      HW_2374P1_Interface_Port_1 { ExternalAccessible := 'False'; ExternalVisible := 'False'; ExternalWritable := 'False'} : HW_INTERFACE := 995;   // "2374P1~Interface~Port_1"
      HW_2374P1_Interface_Port_2 { ExternalAccessible := 'False'; ExternalVisible := 'False'; ExternalWritable := 'False'} : HW_INTERFACE := 996;   // "2374P1~Interface~Port_2"
      HW_2374P1_Head { ExternalAccessible := 'False'; ExternalVisible := 'False'; ExternalWritable := 'False'} : HW_SUBMODULE := 997;   // "2374P1~Head"
      HW_2374P1_EO_Multiturn_1 { ExternalAccessible := 'False'; ExternalVisible := 'False'; ExternalWritable := 'False'} : HW_SUBMODULE := 998;   // "2374P1~EO_Multiturn_1"
      HW_2374P1_Telegram_81_DI_DO { ExternalAccessible := 'False'; ExternalVisible := 'False'; ExternalWritable := 'False'} : HW_SUBMODULE := 999;   // "2374P1_Telegram_81~DI_DO"
      HW_2374P1_EO_Multiturn_1_Parameter_Access_Point { ExternalAccessible := 'False'; ExternalVisible := 'False'; ExternalWritable := 'False'} : HW_SUBMODULE := 1000;   // "2374P1~EO_Multiturn_1~Parameter_Access_Point"
      HW_100A1_Proxy { ExternalAccessible := 'False'; ExternalVisible := 'False'; ExternalWritable := 'False'} : HW_SUBMODULE := 866;   // "100A1~Proxy"
      HW_100A1_IODevice { ExternalAccessible := 'False'; ExternalVisible := 'False'; ExternalWritable := 'False'} : HW_DEVICE := 864;   // "100A1~IODevice"
      HW_100A1_PN_IO { ExternalAccessible := 'False'; ExternalVisible := 'False'; ExternalWritable := 'False'} : HW_INTERFACE := 867;   // "100A1~PN-IO"
      HW_100A1_PN_IO_Port_1 { ExternalAccessible := 'False'; ExternalVisible := 'False'; ExternalWritable := 'False'} : HW_INTERFACE := 868;   // "100A1~PN-IO~Port_1"
      HW_100A1_PN_IO_Port_2 { ExternalAccessible := 'False'; ExternalVisible := 'False'; ExternalWritable := 'False'} : HW_INTERFACE := 869;   // "100A1~PN-IO~Port_2"
      HW_100A1_Head { ExternalAccessible := 'False'; ExternalVisible := 'False'; ExternalWritable := 'False'} : HW_SUBMODULE := 870;   // "100A1~Head"
      HW_2394P1_Proxy { ExternalAccessible := 'False'; ExternalVisible := 'False'; ExternalWritable := 'False'} : HW_SUBMODULE := 1003;   // "2394P1~Proxy"
      HW_2394P1_IODevice { ExternalAccessible := 'False'; ExternalVisible := 'False'; ExternalWritable := 'False'} : HW_DEVICE := 1001;   // "2394P1~IODevice"
      HW_2394P1_Interface { ExternalAccessible := 'False'; ExternalVisible := 'False'; ExternalWritable := 'False'} : HW_INTERFACE := 1004;   // "2394P1~Interface"
      HW_2394P1_Interface_Port_1 { ExternalAccessible := 'False'; ExternalVisible := 'False'; ExternalWritable := 'False'} : HW_INTERFACE := 1005;   // "2394P1~Interface~Port_1"
      HW_2394P1_Interface_Port_2 { ExternalAccessible := 'False'; ExternalVisible := 'False'; ExternalWritable := 'False'} : HW_INTERFACE := 1006;   // "2394P1~Interface~Port_2"
      HW_2394P1_Head { ExternalAccessible := 'False'; ExternalVisible := 'False'; ExternalWritable := 'False'} : HW_SUBMODULE := 1007;   // "2394P1~Head"
      HW_2394P1_EO_Multiturn_1 { ExternalAccessible := 'False'; ExternalVisible := 'False'; ExternalWritable := 'False'} : HW_SUBMODULE := 1008;   // "2394P1~EO_Multiturn_1"
      HW_2394P1_Telegram_81_DI_DO { ExternalAccessible := 'False'; ExternalVisible := 'False'; ExternalWritable := 'False'} : HW_SUBMODULE := 1009;   // "2394P1_Telegram_81~DI_DO"
      HW_2394P1_EO_Multiturn_1_Parameter_Access_Point { ExternalAccessible := 'False'; ExternalVisible := 'False'; ExternalWritable := 'False'} : HW_SUBMODULE := 1010;   // "2394P1~EO_Multiturn_1~Parameter_Access_Point"
      HW_2404P1_Proxy { ExternalAccessible := 'False'; ExternalVisible := 'False'; ExternalWritable := 'False'} : HW_SUBMODULE := 1013;   // "2404P1~Proxy"
      HW_2404P1_IODevice { ExternalAccessible := 'False'; ExternalVisible := 'False'; ExternalWritable := 'False'} : HW_DEVICE := 1011;   // "2404P1~IODevice"
      HW_2404P1_Interface { ExternalAccessible := 'False'; ExternalVisible := 'False'; ExternalWritable := 'False'} : HW_INTERFACE := 1014;   // "2404P1~Interface"
      HW_2404P1_Interface_Port_1 { ExternalAccessible := 'False'; ExternalVisible := 'False'; ExternalWritable := 'False'} : HW_INTERFACE := 1015;   // "2404P1~Interface~Port_1"
      HW_2404P1_Interface_Port_2 { ExternalAccessible := 'False'; ExternalVisible := 'False'; ExternalWritable := 'False'} : HW_INTERFACE := 1016;   // "2404P1~Interface~Port_2"
      HW_2404P1_Head { ExternalAccessible := 'False'; ExternalVisible := 'False'; ExternalWritable := 'False'} : HW_SUBMODULE := 1017;   // "2404P1~Head"
      HW_2404P1_EO_Multiturn_1 { ExternalAccessible := 'False'; ExternalVisible := 'False'; ExternalWritable := 'False'} : HW_SUBMODULE := 1018;   // "2404P1~EO_Multiturn_1"
      HW_2404P1_Telegram_81_DI_DO { ExternalAccessible := 'False'; ExternalVisible := 'False'; ExternalWritable := 'False'} : HW_SUBMODULE := 1019;   // "2404P1_Telegram_81~DI_DO"
      HW_2404P1_EO_Multiturn_1_Parameter_Access_Point { ExternalAccessible := 'False'; ExternalVisible := 'False'; ExternalWritable := 'False'} : HW_SUBMODULE := 1020;   // "2404P1~EO_Multiturn_1~Parameter_Access_Point"
      HW_2434P1_Proxy { ExternalAccessible := 'False'; ExternalVisible := 'False'; ExternalWritable := 'False'} : HW_SUBMODULE := 1023;   // "2434P1~Proxy"
      HW_2434P1_IODevice { ExternalAccessible := 'False'; ExternalVisible := 'False'; ExternalWritable := 'False'} : HW_DEVICE := 1021;   // "2434P1~IODevice"
      HW_2434P1_Interface { ExternalAccessible := 'False'; ExternalVisible := 'False'; ExternalWritable := 'False'} : HW_INTERFACE := 1024;   // "2434P1~Interface"
      HW_2434P1_Interface_Port_1 { ExternalAccessible := 'False'; ExternalVisible := 'False'; ExternalWritable := 'False'} : HW_INTERFACE := 1025;   // "2434P1~Interface~Port_1"
      HW_2434P1_Interface_Port_2 { ExternalAccessible := 'False'; ExternalVisible := 'False'; ExternalWritable := 'False'} : HW_INTERFACE := 1026;   // "2434P1~Interface~Port_2"
      HW_2434P1_Head { ExternalAccessible := 'False'; ExternalVisible := 'False'; ExternalWritable := 'False'} : HW_SUBMODULE := 1027;   // "2434P1~Head"
      HW_2434P1_EO_Multiturn_1 { ExternalAccessible := 'False'; ExternalVisible := 'False'; ExternalWritable := 'False'} : HW_SUBMODULE := 1028;   // "2434P1~EO_Multiturn_1"
      HW_2434P1_Telegram_81_DI_DO { ExternalAccessible := 'False'; ExternalVisible := 'False'; ExternalWritable := 'False'} : HW_SUBMODULE := 1029;   // "2434P1_Telegram_81~DI_DO"
      HW_2434P1_EO_Multiturn_1_Parameter_Access_Point { ExternalAccessible := 'False'; ExternalVisible := 'False'; ExternalWritable := 'False'} : HW_SUBMODULE := 1030;   // "2434P1~EO_Multiturn_1~Parameter_Access_Point"
      HW_2464P1_Proxy { ExternalAccessible := 'False'; ExternalVisible := 'False'; ExternalWritable := 'False'} : HW_SUBMODULE := 1033;   // "2464P1~Proxy"
      HW_2464P1_IODevice { ExternalAccessible := 'False'; ExternalVisible := 'False'; ExternalWritable := 'False'} : HW_DEVICE := 1031;   // "2464P1~IODevice"
      HW_2464P1_Interface { ExternalAccessible := 'False'; ExternalVisible := 'False'; ExternalWritable := 'False'} : HW_INTERFACE := 1034;   // "2464P1~Interface"
      HW_2464P1_Interface_Port_1 { ExternalAccessible := 'False'; ExternalVisible := 'False'; ExternalWritable := 'False'} : HW_INTERFACE := 1035;   // "2464P1~Interface~Port_1"
      HW_2464P1_Interface_Port_2 { ExternalAccessible := 'False'; ExternalVisible := 'False'; ExternalWritable := 'False'} : HW_INTERFACE := 1036;   // "2464P1~Interface~Port_2"
      HW_2464P1_Head { ExternalAccessible := 'False'; ExternalVisible := 'False'; ExternalWritable := 'False'} : HW_SUBMODULE := 1037;   // "2464P1~Head"
      HW_2464P1_EO_Multiturn_1 { ExternalAccessible := 'False'; ExternalVisible := 'False'; ExternalWritable := 'False'} : HW_SUBMODULE := 1038;   // "2464P1~EO_Multiturn_1"
      HW_2464P1_Telegram_81_DI_DO { ExternalAccessible := 'False'; ExternalVisible := 'False'; ExternalWritable := 'False'} : HW_SUBMODULE := 1039;   // "2464P1_Telegram_81~DI_DO"
      HW_2464P1_EO_Multiturn_1_Parameter_Access_Point { ExternalAccessible := 'False'; ExternalVisible := 'False'; ExternalWritable := 'False'} : HW_SUBMODULE := 1040;   // "2464P1~EO_Multiturn_1~Parameter_Access_Point"
      HW_2104P1_Telegram_81_DI_DO : HW_SUBMODULE := 1041;
      HW_2184P1_Telegram_81_DI_DO : HW_SUBMODULE := 824;
      HW_100A1_Voltage_L1_N_1 { ExternalAccessible := 'False'; ExternalVisible := 'False'; ExternalWritable := 'False'} : HW_SUBMODULE := 675;   // "100A1~Voltage_L1-N_1"
      HW_100A1_Voltage_L2_N_1 { ExternalAccessible := 'False'; ExternalVisible := 'False'; ExternalWritable := 'False'} : HW_SUBMODULE := 676;   // "100A1~Voltage_L2-N_1"
      HW_100A1_Voltage_L3_N_1 { ExternalAccessible := 'False'; ExternalVisible := 'False'; ExternalWritable := 'False'} : HW_SUBMODULE := 677;   // "100A1~Voltage_L3-N_1"
      HW_100A1_Current_L1_1 { ExternalAccessible := 'False'; ExternalVisible := 'False'; ExternalWritable := 'False'} : HW_SUBMODULE := 678;   // "100A1~Current_L1_1"
      HW_100A1_Current_L2_1 { ExternalAccessible := 'False'; ExternalVisible := 'False'; ExternalWritable := 'False'} : HW_SUBMODULE := 679;   // "100A1~Current_L2_1"
      HW_100A1_Current_L3_1 { ExternalAccessible := 'False'; ExternalVisible := 'False'; ExternalWritable := 'False'} : HW_SUBMODULE := 680;   // "100A1~Current_L3_1"
      HW_100A1_3_Ph_Average_Volt_L_L_1 { ExternalAccessible := 'False'; ExternalVisible := 'False'; ExternalWritable := 'False'} : HW_SUBMODULE := 681;   // "100A1~3-Ph_Average_Volt_L-L_1"
      HW_100A1_3_Ph_Average_Curr_1 { ExternalAccessible := 'False'; ExternalVisible := 'False'; ExternalWritable := 'False'} : HW_SUBMODULE := 702;   // "100A1~3-Ph_Average_Curr__1"
      HW_100A1_Total_Active_Power_1 { ExternalAccessible := 'False'; ExternalVisible := 'False'; ExternalWritable := 'False'} : HW_SUBMODULE := 705;   // "100A1~Total_Active_Power_1"
      HW_100A1_Total_Reac_Power_1 { ExternalAccessible := 'False'; ExternalVisible := 'False'; ExternalWritable := 'False'} : HW_SUBMODULE := 706;   // "100A1~Total_Reac_Power_1"
      HW_100A1_Act_Energy_Imp_Tar_1_D_1 { ExternalAccessible := 'False'; ExternalVisible := 'False'; ExternalWritable := 'False'} : HW_SUBMODULE := 707;   // "100A1~Act_Energy_Imp_Tar_1(D)_1"
      HW_100A1_Reac_En_Imp_Tar_1_D_1 { ExternalAccessible := 'False'; ExternalVisible := 'False'; ExternalWritable := 'False'} : HW_SUBMODULE := 708;   // "100A1~Reac_En_Imp_Tar_1_(D)_1"
      HW_490A1_JB301_498A1 { ExternalAccessible := 'False'; ExternalVisible := 'False'; ExternalWritable := 'False'} : HW_SUBMODULE := 370;   // "490A1_JB301~498A1"
      HW_490A1_JB301_498A2 { ExternalAccessible := 'False'; ExternalVisible := 'False'; ExternalWritable := 'False'} : HW_SUBMODULE := 371;   // "490A1_JB301~498A2"
      HW_490A1_JB301_498A3 { ExternalAccessible := 'False'; ExternalVisible := 'False'; ExternalWritable := 'False'} : HW_SUBMODULE := 372;   // "490A1_JB301~498A3"
      HW_490A1_JB301_500A1 { ExternalAccessible := 'False'; ExternalVisible := 'False'; ExternalWritable := 'False'} : HW_SUBMODULE := 373;   // "490A1_JB301~500A1"
      HW_490A1_JB301_502A1 { ExternalAccessible := 'False'; ExternalVisible := 'False'; ExternalWritable := 'False'} : HW_SUBMODULE := 374;   // "490A1_JB301~502A1"
      HW_490A1_JB301_502A2 { ExternalAccessible := 'False'; ExternalVisible := 'False'; ExternalWritable := 'False'} : HW_SUBMODULE := 375;   // "490A1_JB301~502A2"
      HW_490A1_JB301_495A3 { ExternalAccessible := 'False'; ExternalVisible := 'False'; ExternalWritable := 'False'} : HW_SUBMODULE := 598;   // "490A1_JB301~495A3"
      CU1_PN_580A1_SIEMENS_telegram_393 { ExternalAccessible := 'False'; ExternalVisible := 'False'; ExternalWritable := 'False'} : HW_SUBMODULE := 709;   // "CU1~PN~580A1_SIEMENS_telegram_393"
      CU1_PN_580A1_SIEMENS_telegram_393_1 { ExternalAccessible := 'False'; ExternalVisible := 'False'; ExternalWritable := 'False'} : HW_SUBMODULE := 709;   // "CU1~PN~580A1_SIEMENS_telegram_393(1)"
      CU1_PN_740A1_1_PROFIsafe_telegram_30 { ExternalAccessible := 'False'; ExternalVisible := 'False'; ExternalWritable := 'False'} : HW_SUBMODULE := 285;   // "CU1~PN~740A1_1_PROFIsafe_telegram_30"
      CU1_PN_740A1_1_PROFIsafe_telegram_30_1 { ExternalAccessible := 'False'; ExternalVisible := 'False'; ExternalWritable := 'False'} : HW_SUBMODULE := 285;   // "CU1~PN~740A1_1_PROFIsafe_telegram_30(1)"
      CU1_PN_740A1_2_PROFIsafe_telegram_30 { ExternalAccessible := 'False'; ExternalVisible := 'False'; ExternalWritable := 'False'} : HW_SUBMODULE := 319;   // "CU1~PN~740A1_2_PROFIsafe_telegram_30"
      CU1_PN_740A1_2_PROFIsafe_telegram_30_1 { ExternalAccessible := 'False'; ExternalVisible := 'False'; ExternalWritable := 'False'} : HW_SUBMODULE := 319;   // "CU1~PN~740A1_2_PROFIsafe_telegram_30(1)"
      CU1_PN_690A1_1_PROFIsafe_telegram_30 { ExternalAccessible := 'False'; ExternalVisible := 'False'; ExternalWritable := 'False'} : HW_SUBMODULE := 460;   // "CU1~PN~690A1_1_PROFIsafe_telegram_30"
      CU1_PN_690A1_1_PROFIsafe_telegram_30_1 { ExternalAccessible := 'False'; ExternalVisible := 'False'; ExternalWritable := 'False'} : HW_SUBMODULE := 460;   // "CU1~PN~690A1_1_PROFIsafe_telegram_30(1)"
      CU1_PN_690A1_2_PROFIsafe_telegram_30 { ExternalAccessible := 'False'; ExternalVisible := 'False'; ExternalWritable := 'False'} : HW_SUBMODULE := 464;   // "CU1~PN~690A1_2_PROFIsafe_telegram_30"
      CU1_PN_690A1_2_PROFIsafe_telegram_30_1 { ExternalAccessible := 'False'; ExternalVisible := 'False'; ExternalWritable := 'False'} : HW_SUBMODULE := 464;   // "CU1~PN~690A1_2_PROFIsafe_telegram_30(1)"
      CU1_PN_890A1_1_PROFIsafe_telegram_30 { ExternalAccessible := 'False'; ExternalVisible := 'False'; ExternalWritable := 'False'} : HW_SUBMODULE := 468;   // "CU1~PN~890A1_1_PROFIsafe_telegram_30"
      CU1_PN_890A1_1_PROFIsafe_telegram_30_1 { ExternalAccessible := 'False'; ExternalVisible := 'False'; ExternalWritable := 'False'} : HW_SUBMODULE := 468;   // "CU1~PN~890A1_1_PROFIsafe_telegram_30(1)"
      CU1_PN_890A1_2_PROFIsafe_telegram_30 { ExternalAccessible := 'False'; ExternalVisible := 'False'; ExternalWritable := 'False'} : HW_SUBMODULE := 472;   // "CU1~PN~890A1_2_PROFIsafe_telegram_30"
      CU1_PN_890A1_2_PROFIsafe_telegram_30_1 { ExternalAccessible := 'False'; ExternalVisible := 'False'; ExternalWritable := 'False'} : HW_SUBMODULE := 472;   // "CU1~PN~890A1_2_PROFIsafe_telegram_30(1)"
      HW_490A1_JB301_Server_module_1 { ExternalAccessible := 'False'; ExternalVisible := 'False'; ExternalWritable := 'False'} : HW_SUBMODULE := 473;   // "490A1_JB301~Server_module_1"
      HW_510A1_JB302_518A1 { ExternalAccessible := 'False'; ExternalVisible := 'False'; ExternalWritable := 'False'} : HW_SUBMODULE := 387;   // "510A1_JB302~518A1"
      HW_510A1_JB302_518A2 { ExternalAccessible := 'False'; ExternalVisible := 'False'; ExternalWritable := 'False'} : HW_SUBMODULE := 388;   // "510A1_JB302~518A2"
      HW_510A1_JB302_518A3 { ExternalAccessible := 'False'; ExternalVisible := 'False'; ExternalWritable := 'False'} : HW_SUBMODULE := 389;   // "510A1_JB302~518A3"
      HW_510A1_JB302_518A4 { ExternalAccessible := 'False'; ExternalVisible := 'False'; ExternalWritable := 'False'} : HW_SUBMODULE := 390;   // "510A1_JB302~518A4"
      HW_510A1_JB302_518A5 { ExternalAccessible := 'False'; ExternalVisible := 'False'; ExternalWritable := 'False'} : HW_SUBMODULE := 391;   // "510A1_JB302~518A5"
      HW_510A1_JB302_518A6 { ExternalAccessible := 'False'; ExternalVisible := 'False'; ExternalWritable := 'False'} : HW_SUBMODULE := 392;   // "510A1_JB302~518A6"
      HW_510A1_JB302_518A7 { ExternalAccessible := 'False'; ExternalVisible := 'False'; ExternalWritable := 'False'} : HW_SUBMODULE := 393;   // "510A1_JB302~518A7"
      HW_510A1_JB302_518A8 { ExternalAccessible := 'False'; ExternalVisible := 'False'; ExternalWritable := 'False'} : HW_SUBMODULE := 394;   // "510A1_JB302~518A8"
      HW_510A1_JB302_519A1 { ExternalAccessible := 'False'; ExternalVisible := 'False'; ExternalWritable := 'False'} : HW_SUBMODULE := 395;   // "510A1_JB302~519A1"
      HW_510A1_JB302_519A2 { ExternalAccessible := 'False'; ExternalVisible := 'False'; ExternalWritable := 'False'} : HW_SUBMODULE := 396;   // "510A1_JB302~519A2"
      HW_510A1_JB302_519A3 { ExternalAccessible := 'False'; ExternalVisible := 'False'; ExternalWritable := 'False'} : HW_SUBMODULE := 397;   // "510A1_JB302~519A3"
      HW_510A1_JB302_519A4 { ExternalAccessible := 'False'; ExternalVisible := 'False'; ExternalWritable := 'False'} : HW_SUBMODULE := 398;   // "510A1_JB302~519A4"
      HW_510A1_JB302_519A5 { ExternalAccessible := 'False'; ExternalVisible := 'False'; ExternalWritable := 'False'} : HW_SUBMODULE := 399;   // "510A1_JB302~519A5"
      HW_510A1_JB302_520A1 { ExternalAccessible := 'False'; ExternalVisible := 'False'; ExternalWritable := 'False'} : HW_SUBMODULE := 400;   // "510A1_JB302~520A1"
      HW_510A1_JB302_520A2 { ExternalAccessible := 'False'; ExternalVisible := 'False'; ExternalWritable := 'False'} : HW_SUBMODULE := 401;   // "510A1_JB302~520A2"
      HW_510A1_JB302_522A1 { ExternalAccessible := 'False'; ExternalVisible := 'False'; ExternalWritable := 'False'} : HW_SUBMODULE := 402;   // "510A1_JB302~522A1"
      HW_510A1_JB302_522A2 { ExternalAccessible := 'False'; ExternalVisible := 'False'; ExternalWritable := 'False'} : HW_SUBMODULE := 403;   // "510A1_JB302~522A2"
      HW_510A1_JB302_522A3 { ExternalAccessible := 'False'; ExternalVisible := 'False'; ExternalWritable := 'False'} : HW_SUBMODULE := 404;   // "510A1_JB302~522A3"
      HW_510A1_JB302_522A4 { ExternalAccessible := 'False'; ExternalVisible := 'False'; ExternalWritable := 'False'} : HW_SUBMODULE := 405;   // "510A1_JB302~522A4"
      HW_510A1_JB302_522A5 { ExternalAccessible := 'False'; ExternalVisible := 'False'; ExternalWritable := 'False'} : HW_SUBMODULE := 406;   // "510A1_JB302~522A5"
      HW_510A1_JB302_522A6 { ExternalAccessible := 'False'; ExternalVisible := 'False'; ExternalWritable := 'False'} : HW_SUBMODULE := 407;   // "510A1_JB302~522A6"
      HW_510A1_JB302_522A7 { ExternalAccessible := 'False'; ExternalVisible := 'False'; ExternalWritable := 'False'} : HW_SUBMODULE := 408;   // "510A1_JB302~522A7"
      HW_510A1_JB302_522A8 { ExternalAccessible := 'False'; ExternalVisible := 'False'; ExternalWritable := 'False'} : HW_SUBMODULE := 409;   // "510A1_JB302~522A8"
      HW_510A1_JB302_Server_module_1 { ExternalAccessible := 'False'; ExternalVisible := 'False'; ExternalWritable := 'False'} : HW_SUBMODULE := 410;   // "510A1_JB302~Server_module_1"
      HW_530A1_JB305_Server_module_1 { ExternalAccessible := 'False'; ExternalVisible := 'False'; ExternalWritable := 'False'} : HW_SUBMODULE := 596;   // "530A1_JB305~Server_module_1"
      HW_530A1_JB305_532A1 { ExternalAccessible := 'False'; ExternalVisible := 'False'; ExternalWritable := 'False'} : HW_SUBMODULE := 418;   // "530A1_JB305~532A1"
      HW_550A1_JB306_Server_module_1 { ExternalAccessible := 'False'; ExternalVisible := 'False'; ExternalWritable := 'False'} : HW_SUBMODULE := 595;   // "550A1_JB306~Server_module_1"
      HU_Cytropac_Proxy { ExternalAccessible := 'False'; ExternalVisible := 'False'; ExternalWritable := 'False'} : HW_SUBMODULE := 711;   // "HU_Cytropac~Proxy"
      HU_Cytropac_IODevice { ExternalAccessible := 'False'; ExternalVisible := 'False'; ExternalWritable := 'False'} : HW_DEVICE := 597;   // "HU_Cytropac~IODevice"
      HU_Cytropac_PN_IO { ExternalAccessible := 'False'; ExternalVisible := 'False'; ExternalWritable := 'False'} : HW_INTERFACE := 712;   // "HU_Cytropac~PN-IO"
      HU_Cytropac_PN_IO_Port_1_RJ45 { ExternalAccessible := 'False'; ExternalVisible := 'False'; ExternalWritable := 'False'} : HW_INTERFACE := 713;   // "HU_Cytropac~PN-IO~Port_1_-_RJ45"
      HU_Cytropac_PN_IO_Port_2_RJ45 { ExternalAccessible := 'False'; ExternalVisible := 'False'; ExternalWritable := 'False'} : HW_INTERFACE := 714;   // "HU_Cytropac~PN-IO~Port_2_-_RJ45"
      HU_Cytropac_Head { ExternalAccessible := 'False'; ExternalVisible := 'False'; ExternalWritable := 'False'} : HW_SUBMODULE := 715;   // "HU_Cytropac~Head"
      HU_Cytropac_Output_04_Words_1 { ExternalAccessible := 'False'; ExternalVisible := 'False'; ExternalWritable := 'False'} : HW_SUBMODULE := 716;   // "HU_Cytropac~Output_04_Words_1"
      HU_Cytropac_Input_08_Words_1 { ExternalAccessible := 'False'; ExternalVisible := 'False'; ExternalWritable := 'False'} : HW_SUBMODULE := 717;   // "HU_Cytropac~Input_08_Words_1"
      CU1_PN_740A1_1_Standard_telegram_1 { ExternalAccessible := 'False'; ExternalVisible := 'False'; ExternalWritable := 'False'} : HW_SUBMODULE := 282;   // "CU1~PN~740A1_1_Standard_telegram_1"
      CU1_PN_740A1_1_Standard_telegram_1_1 { ExternalAccessible := 'False'; ExternalVisible := 'False'; ExternalWritable := 'False'} : HW_SUBMODULE := 282;   // "CU1~PN~740A1_1_Standard_telegram_1(1)"
      CU1_PN_740A1_2_Standard_telegram_1 { ExternalAccessible := 'False'; ExternalVisible := 'False'; ExternalWritable := 'False'} : HW_SUBMODULE := 286;   // "CU1~PN~740A1_2_Standard_telegram_1"
      CU1_PN_740A1_2_Standard_telegram_1_1 { ExternalAccessible := 'False'; ExternalVisible := 'False'; ExternalWritable := 'False'} : HW_SUBMODULE := 286;   // "CU1~PN~740A1_2_Standard_telegram_1(1)"
      CU1_PN_690A1_1_Standard_telegram_1 { ExternalAccessible := 'False'; ExternalVisible := 'False'; ExternalWritable := 'False'} : HW_SUBMODULE := 457;   // "CU1~PN~690A1_1_Standard_telegram_1"
      CU1_PN_690A1_1_Standard_telegram_1_1 { ExternalAccessible := 'False'; ExternalVisible := 'False'; ExternalWritable := 'False'} : HW_SUBMODULE := 457;   // "CU1~PN~690A1_1_Standard_telegram_1(1)"
      CU1_PN_690A1_2_Standard_telegram_1 { ExternalAccessible := 'False'; ExternalVisible := 'False'; ExternalWritable := 'False'} : HW_SUBMODULE := 461;   // "CU1~PN~690A1_2_Standard_telegram_1"
      CU1_PN_690A1_2_Standard_telegram_1_1 { ExternalAccessible := 'False'; ExternalVisible := 'False'; ExternalWritable := 'False'} : HW_SUBMODULE := 461;   // "CU1~PN~690A1_2_Standard_telegram_1(1)"
      CU1_PN_890A1_1_Standard_telegram_1 { ExternalAccessible := 'False'; ExternalVisible := 'False'; ExternalWritable := 'False'} : HW_SUBMODULE := 465;   // "CU1~PN~890A1_1_Standard_telegram_1"
      CU1_PN_890A1_1_Standard_telegram_1_1 { ExternalAccessible := 'False'; ExternalVisible := 'False'; ExternalWritable := 'False'} : HW_SUBMODULE := 465;   // "CU1~PN~890A1_1_Standard_telegram_1(1)"
      CU1_PN_890A1_2_Standard_telegram_1 { ExternalAccessible := 'False'; ExternalVisible := 'False'; ExternalWritable := 'False'} : HW_SUBMODULE := 469;   // "CU1~PN~890A1_2_Standard_telegram_1"
      CU1_PN_890A1_2_Standard_telegram_1_1 { ExternalAccessible := 'False'; ExternalVisible := 'False'; ExternalWritable := 'False'} : HW_SUBMODULE := 469;   // "CU1~PN~890A1_2_Standard_telegram_1(1)"
      CU3_PROFINET_interface_1410A1_1_Standard_telegram_1 { ExternalAccessible := 'False'; ExternalVisible := 'False'; ExternalWritable := 'False'} : HW_SUBMODULE := 485;   // "CU3~PROFINET_interface~1410A1_1_Standard_telegram_1"
      CU3_PROFINET_interface_1410A1_1_Standard_telegram_1_1 { ExternalAccessible := 'False'; ExternalVisible := 'False'; ExternalWritable := 'False'} : HW_SUBMODULE := 485;   // "CU3~PROFINET_interface~1410A1_1_Standard_telegram_1(1)"
      CU3_PROFINET_interface_1410A1_2_Standard_telegram_1 { ExternalAccessible := 'False'; ExternalVisible := 'False'; ExternalWritable := 'False'} : HW_SUBMODULE := 489;   // "CU3~PROFINET_interface~1410A1_2_Standard_telegram_1"
      CU3_PROFINET_interface_1410A1_2_Standard_telegram_1_1 { ExternalAccessible := 'False'; ExternalVisible := 'False'; ExternalWritable := 'False'} : HW_SUBMODULE := 489;   // "CU3~PROFINET_interface~1410A1_2_Standard_telegram_1(1)"
      CU3_PROFINET_interface_1430A1_1_Standard_telegram_1 { ExternalAccessible := 'False'; ExternalVisible := 'False'; ExternalWritable := 'False'} : HW_SUBMODULE := 493;   // "CU3~PROFINET_interface~1430A1_1_Standard_telegram_1"
      CU3_PROFINET_interface_1430A1_1_Standard_telegram_1_1 { ExternalAccessible := 'False'; ExternalVisible := 'False'; ExternalWritable := 'False'} : HW_SUBMODULE := 493;   // "CU3~PROFINET_interface~1430A1_1_Standard_telegram_1(1)"
      CU3_PROFINET_interface_1430A1_2_Standard_telegram_1 { ExternalAccessible := 'False'; ExternalVisible := 'False'; ExternalWritable := 'False'} : HW_SUBMODULE := 497;   // "CU3~PROFINET_interface~1430A1_2_Standard_telegram_1"
      CU3_PROFINET_interface_1430A1_2_Standard_telegram_1_1 { ExternalAccessible := 'False'; ExternalVisible := 'False'; ExternalWritable := 'False'} : HW_SUBMODULE := 497;   // "CU3~PROFINET_interface~1430A1_2_Standard_telegram_1(1)"
      CU3_PROFINET_interface_1260A1_1_Standard_telegram_1 { ExternalAccessible := 'False'; ExternalVisible := 'False'; ExternalWritable := 'False'} : HW_SUBMODULE := 501;   // "CU3~PROFINET_interface~1260A1_1_Standard_telegram_1"
      CU3_PROFINET_interface_1260A1_1_Standard_telegram_1_1 { ExternalAccessible := 'False'; ExternalVisible := 'False'; ExternalWritable := 'False'} : HW_SUBMODULE := 501;   // "CU3~PROFINET_interface~1260A1_1_Standard_telegram_1(1)"
      CU3_PROFINET_interface_1260A1_2_Standard_telegram_1 { ExternalAccessible := 'False'; ExternalVisible := 'False'; ExternalWritable := 'False'} : HW_SUBMODULE := 505;   // "CU3~PROFINET_interface~1260A1_2_Standard_telegram_1"
      CU3_PROFINET_interface_1260A1_2_Standard_telegram_1_1 { ExternalAccessible := 'False'; ExternalVisible := 'False'; ExternalWritable := 'False'} : HW_SUBMODULE := 505;   // "CU3~PROFINET_interface~1260A1_2_Standard_telegram_1(1)"
      CU4_PN_980A1_1_Standard_telegram_1 { ExternalAccessible := 'False'; ExternalVisible := 'False'; ExternalWritable := 'False'} : HW_SUBMODULE := 518;   // "CU4~PN~980A1_1_Standard_telegram_1"
      CU4_PN_980A1_1_Standard_telegram_1_1 { ExternalAccessible := 'False'; ExternalVisible := 'False'; ExternalWritable := 'False'} : HW_SUBMODULE := 518;   // "CU4~PN~980A1_1_Standard_telegram_1(1)"
      CU4_PN_980A1_2_Standard_telegram_1 { ExternalAccessible := 'False'; ExternalVisible := 'False'; ExternalWritable := 'False'} : HW_SUBMODULE := 522;   // "CU4~PN~980A1_2_Standard_telegram_1"
      CU4_PN_980A1_2_Standard_telegram_1_1 { ExternalAccessible := 'False'; ExternalVisible := 'False'; ExternalWritable := 'False'} : HW_SUBMODULE := 522;   // "CU4~PN~980A1_2_Standard_telegram_1(1)"
      CU4_PN_1030A1_1_Standard_telegram_1 { ExternalAccessible := 'False'; ExternalVisible := 'False'; ExternalWritable := 'False'} : HW_SUBMODULE := 526;   // "CU4~PN~1030A1_1_Standard_telegram_1"
      CU4_PN_1030A1_1_Standard_telegram_1_1 { ExternalAccessible := 'False'; ExternalVisible := 'False'; ExternalWritable := 'False'} : HW_SUBMODULE := 526;   // "CU4~PN~1030A1_1_Standard_telegram_1(1)"
      CU4_PN_1030A1_2_Standard_telegram_1 { ExternalAccessible := 'False'; ExternalVisible := 'False'; ExternalWritable := 'False'} : HW_SUBMODULE := 530;   // "CU4~PN~1030A1_2_Standard_telegram_1"
      CU4_PN_1030A1_2_Standard_telegram_1_1 { ExternalAccessible := 'False'; ExternalVisible := 'False'; ExternalWritable := 'False'} : HW_SUBMODULE := 530;   // "CU4~PN~1030A1_2_Standard_telegram_1(1)"
      CU4_PN_1070A1_1_Standard_telegram_1 { ExternalAccessible := 'False'; ExternalVisible := 'False'; ExternalWritable := 'False'} : HW_SUBMODULE := 534;   // "CU4~PN~1070A1_1_Standard_telegram_1"
      CU4_PN_1070A1_1_Standard_telegram_1_1 { ExternalAccessible := 'False'; ExternalVisible := 'False'; ExternalWritable := 'False'} : HW_SUBMODULE := 534;   // "CU4~PN~1070A1_1_Standard_telegram_1(1)"
      CU4_PN_1070A1_2_Standard_telegram_1 { ExternalAccessible := 'False'; ExternalVisible := 'False'; ExternalWritable := 'False'} : HW_SUBMODULE := 538;   // "CU4~PN~1070A1_2_Standard_telegram_1"
      CU4_PN_1070A1_2_Standard_telegram_1_1 { ExternalAccessible := 'False'; ExternalVisible := 'False'; ExternalWritable := 'False'} : HW_SUBMODULE := 538;   // "CU4~PN~1070A1_2_Standard_telegram_1(1)"
      CU5_PN_1480A1_1_Standard_telegram_1 { ExternalAccessible := 'False'; ExternalVisible := 'False'; ExternalWritable := 'False'} : HW_SUBMODULE := 555;   // "CU5~PN~1480A1_1_Standard_telegram_1"
      CU5_PN_1480A1_1_Standard_telegram_1_1 { ExternalAccessible := 'False'; ExternalVisible := 'False'; ExternalWritable := 'False'} : HW_SUBMODULE := 555;   // "CU5~PN~1480A1_1_Standard_telegram_1(1)"
      CU5_PN_1480A1_2_Standard_telegram_1 { ExternalAccessible := 'False'; ExternalVisible := 'False'; ExternalWritable := 'False'} : HW_SUBMODULE := 559;   // "CU5~PN~1480A1_2_Standard_telegram_1"
      CU5_PN_1480A1_2_Standard_telegram_1_1 { ExternalAccessible := 'False'; ExternalVisible := 'False'; ExternalWritable := 'False'} : HW_SUBMODULE := 559;   // "CU5~PN~1480A1_2_Standard_telegram_1(1)"
      CU5_PN_1560A1_2_Standard_telegram_1_2 { ExternalAccessible := 'False'; ExternalVisible := 'False'; ExternalWritable := 'False'} : HW_SUBMODULE := 567;
      CU6_PN_1990A1_1_Standard_telegram_1 { ExternalAccessible := 'False'; ExternalVisible := 'False'; ExternalWritable := 'False'} : HW_SUBMODULE := 580;   // "CU6~PN~1990A1_1_Standard_telegram_1"
      CU6_PN_1990A1_1_Standard_telegram_1_1 { ExternalAccessible := 'False'; ExternalVisible := 'False'; ExternalWritable := 'False'} : HW_SUBMODULE := 580;   // "CU6~PN~1990A1_1_Standard_telegram_1(1)"
      CU6_PN_1990A1_2_Standard_telegram_1 { ExternalAccessible := 'False'; ExternalVisible := 'False'; ExternalWritable := 'False'} : HW_SUBMODULE := 584;   // "CU6~PN~1990A1_2_Standard_telegram_1"
      CU6_PN_1990A1_2_Standard_telegram_1_1 { ExternalAccessible := 'False'; ExternalVisible := 'False'; ExternalWritable := 'False'} : HW_SUBMODULE := 584;   // "CU6~PN~1990A1_2_Standard_telegram_1(1)"
      CU6_PN_1840A1_1_Standard_telegram_1 { ExternalAccessible := 'False'; ExternalVisible := 'False'; ExternalWritable := 'False'} : HW_SUBMODULE := 600;   // "CU6~PN~1840A1_1_Standard_telegram_1"
      CU6_PN_1840A1_1_Standard_telegram_1_1 { ExternalAccessible := 'False'; ExternalVisible := 'False'; ExternalWritable := 'False'} : HW_SUBMODULE := 600;   // "CU6~PN~1840A1_1_Standard_telegram_1(1)"
      CU6_PN_1840A1_2_Standard_telegram_1 { ExternalAccessible := 'False'; ExternalVisible := 'False'; ExternalWritable := 'False'} : HW_SUBMODULE := 604;   // "CU6~PN~1840A1_2_Standard_telegram_1"
      CU6_PN_1840A1_2_Standard_telegram_1_1 { ExternalAccessible := 'False'; ExternalVisible := 'False'; ExternalWritable := 'False'} : HW_SUBMODULE := 604;   // "CU6~PN~1840A1_2_Standard_telegram_1(1)"
      CU7_PN_2260A1_1_Standard_telegram_1 { ExternalAccessible := 'False'; ExternalVisible := 'False'; ExternalWritable := 'False'} : HW_SUBMODULE := 625;   // "CU7~PN~2260A1_1_Standard_telegram_1"
      CU7_PN_2260A1_1_Standard_telegram_1_1 { ExternalAccessible := 'False'; ExternalVisible := 'False'; ExternalWritable := 'False'} : HW_SUBMODULE := 625;   // "CU7~PN~2260A1_1_Standard_telegram_1(1)"
      CU7_PN_2260A1_2_Standard_telegram_1 { ExternalAccessible := 'False'; ExternalVisible := 'False'; ExternalWritable := 'False'} : HW_SUBMODULE := 629;   // "CU7~PN~2260A1_2_Standard_telegram_1"
      CU7_PN_2260A1_2_Standard_telegram_1_1 { ExternalAccessible := 'False'; ExternalVisible := 'False'; ExternalWritable := 'False'} : HW_SUBMODULE := 629;   // "CU7~PN~2260A1_2_Standard_telegram_1(1)"
      CU8_PN_2390A1_1_Standard_telegram_1 { ExternalAccessible := 'False'; ExternalVisible := 'False'; ExternalWritable := 'False'} : HW_SUBMODULE := 651;   // "CU8~PN~2390A1_1_Standard_telegram_1"
      CU8_PN_2390A1_1_Standard_telegram_1_1 { ExternalAccessible := 'False'; ExternalVisible := 'False'; ExternalWritable := 'False'} : HW_SUBMODULE := 651;   // "CU8~PN~2390A1_1_Standard_telegram_1(1)"
      CU8_PN_2390A1_2_Standard_telegram_1 { ExternalAccessible := 'False'; ExternalVisible := 'False'; ExternalWritable := 'False'} : HW_SUBMODULE := 655;   // "CU8~PN~2390A1_2_Standard_telegram_1"
      CU8_PN_2390A1_2_Standard_telegram_1_1 { ExternalAccessible := 'False'; ExternalVisible := 'False'; ExternalWritable := 'False'} : HW_SUBMODULE := 655;   // "CU8~PN~2390A1_2_Standard_telegram_1(1)"
      CU8_PN_2430A1_1_Standard_telegram_1 { ExternalAccessible := 'False'; ExternalVisible := 'False'; ExternalWritable := 'False'} : HW_SUBMODULE := 659;   // "CU8~PN~2430A1_1_Standard_telegram_1"
      CU8_PN_2430A1_1_Standard_telegram_1_1 { ExternalAccessible := 'False'; ExternalVisible := 'False'; ExternalWritable := 'False'} : HW_SUBMODULE := 659;   // "CU8~PN~2430A1_1_Standard_telegram_1(1)"
      CU8_PN_2430A1_2_Standard_telegram_1 { ExternalAccessible := 'False'; ExternalVisible := 'False'; ExternalWritable := 'False'} : HW_SUBMODULE := 663;   // "CU8~PN~2430A1_2_Standard_telegram_1"
      CU8_PN_2430A1_2_Standard_telegram_1_1 { ExternalAccessible := 'False'; ExternalVisible := 'False'; ExternalWritable := 'False'} : HW_SUBMODULE := 663;   // "CU8~PN~2430A1_2_Standard_telegram_1(1)"
      CU8_PN_2350A1_1_Standard_telegram_1 { ExternalAccessible := 'False'; ExternalVisible := 'False'; ExternalWritable := 'False'} : HW_SUBMODULE := 667;   // "CU8~PN~2350A1_1_Standard_telegram_1"
      CU8_PN_2350A1_1_Standard_telegram_1_1 { ExternalAccessible := 'False'; ExternalVisible := 'False'; ExternalWritable := 'False'} : HW_SUBMODULE := 667;   // "CU8~PN~2350A1_1_Standard_telegram_1(1)"
      CU8_PN_2350A1_2_Standard_telegram_1 { ExternalAccessible := 'False'; ExternalVisible := 'False'; ExternalWritable := 'False'} : HW_SUBMODULE := 671;   // "CU8~PN~2350A1_2_Standard_telegram_1"
      CU8_PN_2350A1_2_Standard_telegram_1_1 { ExternalAccessible := 'False'; ExternalVisible := 'False'; ExternalWritable := 'False'} : HW_SUBMODULE := 671;   // "CU8~PN~2350A1_2_Standard_telegram_1(1)"
      CU2_PN_585A1_SIEMENS_telegram_393 { ExternalAccessible := 'False'; ExternalVisible := 'False'; ExternalWritable := 'False'} : HW_SUBMODULE := 274;   // "CU2~PN~585A1_SIEMENS_telegram_393"
      CU2_PN_585A1_SIEMENS_telegram_393_1 { ExternalAccessible := 'False'; ExternalVisible := 'False'; ExternalWritable := 'False'} : HW_SUBMODULE := 274;   // "CU2~PN~585A1_SIEMENS_telegram_393(1)"
      CU2_PN_1190A1_SIEMENS_telegram_106 { ExternalAccessible := 'False'; ExternalVisible := 'False'; ExternalWritable := 'False'} : HW_SUBMODULE := 290;   // "CU2~PN~1190A1_SIEMENS_telegram_106"
      CU2_PN_1190A1_SIEMENS_telegram_106_1 { ExternalAccessible := 'False'; ExternalVisible := 'False'; ExternalWritable := 'False'} : HW_SUBMODULE := 290;   // "CU2~PN~1190A1_SIEMENS_telegram_106(1)"
      CU2_PN_1190A1_PROFIsafe_telegram_30 { ExternalAccessible := 'False'; ExternalVisible := 'False'; ExternalWritable := 'False'} : HW_SUBMODULE := 291;   // "CU2~PN~1190A1_PROFIsafe_telegram_30"
      CU2_PN_1190A1_PROFIsafe_telegram_30_1 { ExternalAccessible := 'False'; ExternalVisible := 'False'; ExternalWritable := 'False'} : HW_SUBMODULE := 291;   // "CU2~PN~1190A1_PROFIsafe_telegram_30(1)"
      CU2_PN_1300A1_SIEMENS_telegram_106 { ExternalAccessible := 'False'; ExternalVisible := 'False'; ExternalWritable := 'False'} : HW_SUBMODULE := 294;   // "CU2~PN~1300A1_SIEMENS_telegram_106"
      CU2_PN_1300A1_SIEMENS_telegram_106_1 { ExternalAccessible := 'False'; ExternalVisible := 'False'; ExternalWritable := 'False'} : HW_SUBMODULE := 294;   // "CU2~PN~1300A1_SIEMENS_telegram_106(1)"
      CU2_PN_1300A1_PROFIsafe_telegram_30 { ExternalAccessible := 'False'; ExternalVisible := 'False'; ExternalWritable := 'False'} : HW_SUBMODULE := 295;   // "CU2~PN~1300A1_PROFIsafe_telegram_30"
      CU2_PN_1300A1_PROFIsafe_telegram_30_1 { ExternalAccessible := 'False'; ExternalVisible := 'False'; ExternalWritable := 'False'} : HW_SUBMODULE := 295;   // "CU2~PN~1300A1_PROFIsafe_telegram_30(1)"
      CU2_PN_830A1_SIEMENS_telegram_106 { ExternalAccessible := 'False'; ExternalVisible := 'False'; ExternalWritable := 'False'} : HW_SUBMODULE := 298;   // "CU2~PN~830A1_SIEMENS_telegram_106"
      CU2_PN_830A1_SIEMENS_telegram_106_1 { ExternalAccessible := 'False'; ExternalVisible := 'False'; ExternalWritable := 'False'} : HW_SUBMODULE := 298;   // "CU2~PN~830A1_SIEMENS_telegram_106(1)"
      CU2_PN_830A1_PROFIsafe_telegram_30 { ExternalAccessible := 'False'; ExternalVisible := 'False'; ExternalWritable := 'False'} : HW_SUBMODULE := 299;   // "CU2~PN~830A1_PROFIsafe_telegram_30"
      CU2_PN_830A1_PROFIsafe_telegram_30_1 { ExternalAccessible := 'False'; ExternalVisible := 'False'; ExternalWritable := 'False'} : HW_SUBMODULE := 299;   // "CU2~PN~830A1_PROFIsafe_telegram_30(1)"
      CU6_PN_2100A1_1_Standard_telegram_1 { ExternalAccessible := 'False'; ExternalVisible := 'False'; ExternalWritable := 'False'} : HW_SUBMODULE := 592;   // "CU8~PN~2390A1_2_Standard_telegram_1"
      CU6_PN_2100A1_2_Standard_telegram_1 { ExternalAccessible := 'False'; ExternalVisible := 'False'; ExternalWritable := 'False'} : HW_SUBMODULE := 588;   // "CU8~PN~2390A1_2_Standard_telegram_1"
      "dl-pn1_DL_PN1_1" { ExternalAccessible := 'False'; ExternalVisible := 'False'; ExternalWritable := 'False'} : HW_SUBMODULE := 784;   // "dl-pn1~DL-PN1_1"
      "dl-pn1_IL-1000_Master" { ExternalAccessible := 'False'; ExternalVisible := 'False'; ExternalWritable := 'False'} : HW_SUBMODULE := 1042;   // dl-pn1~IL-1000_Master
      "dl-pn1_IL-1000_Slave" { ExternalAccessible := 'False'; ExternalVisible := 'False'; ExternalWritable := 'False'} : HW_SUBMODULE := 1043;   // dl-pn1~IL-1050_Salve
   END_VAR
BEGIN
END_DATA_BLOCK
